RoboDK station: MESA_EJEMPLO.rdk

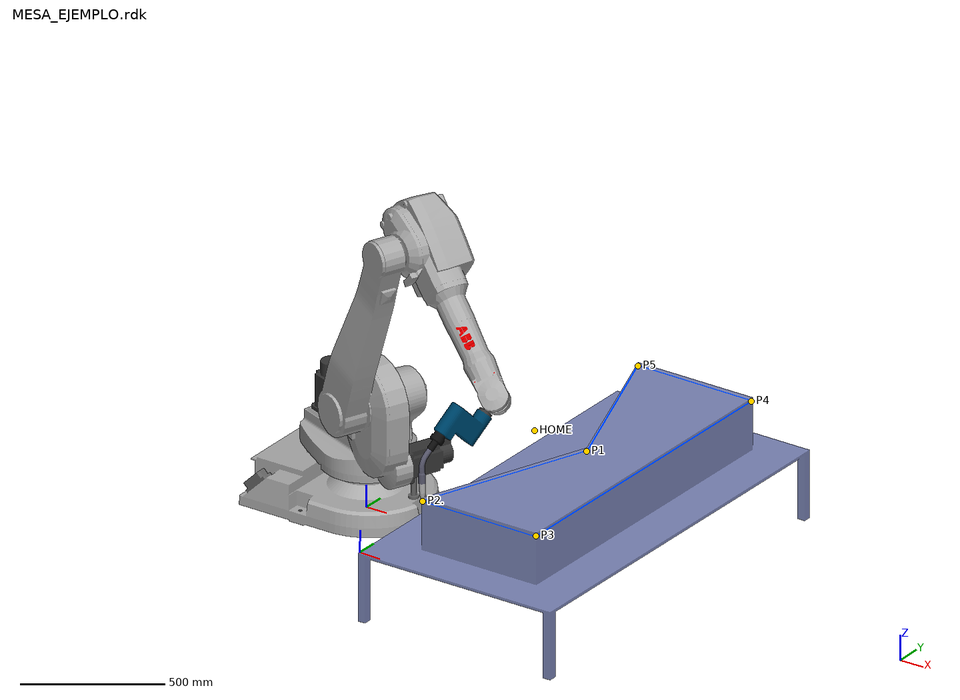
[picture v0: the station drawn from its stored meshes, robots at their saved joint values, targets as dots, program paths as lines]
Station MESA_EJEMPLO (saved by RoboDK 5.9.0). Poses are relative to the parent item; angles as X-Y-Z fixed-axis rotations.
  - frame ABB IRB 1600-6/1.45 Base at (0, 0, 0) mm
    - robot ABB IRB 1600-6/1.45: 6 axes, payload 6 kg, reach 1450 mm, repeatability 0.05 mm, weight 250 kg
        modified DH rows (alpha deg, a mm, theta deg, d mm): 0, 0, 0, 486.5; -90, 150, -90, 0; 0, 700, 0, 0; -90, 0, 0, 600; 90, 0, 0, 0; -90, 0, 180, 65
        joint limits [-180, -90, -245, -200, -115, -400] to [180, 120, 65, 200, 115, 400]; home [0, 0, 0, 0, 0, 0]; saved at [-21.7, 18.023, 24.268, -55.937, 59.398, 126.175]
      - tool Weld gun, TCP at (-4, 0, 371.3) mm, rotated rx 0 ry 45 rz 0 deg, size 299.9 x 60 x 318.3 mm
  - object mesa_ejemplo at (1300, -750, 0) mm, rotated rx 90 ry 0 rz 90 deg, size 1560 x 460 x 810 mm, geometry from mesa_ejemplo.IGS
  - frame Frame 2 at (500.14, -751.72, 267.07) mm, rotated rx -0.99 ry 1.63 rz 0.01 deg
    - target HOME (Cartesian target) at (159.13, 815.13, 203.86) mm, rotated rx 179.01 ry -0.28 rz 179.99 deg; joints [10.42, -21.045, 59.328, -38.186, 11.528, 45.27] of ABB IRB 1600-6/1.45
    - target P1 (Cartesian target) at (390.95, 796.79, 204.49) mm, rotated rx 179.01 ry -0.28 rz 179.99 deg; joints [4.664, 1.836, 43.09, -56.828, 3.804, 60.18] of ABB IRB 1600-6/1.45
    - target P2. (Cartesian target) at (152.66, 148.82, 186.18) mm, rotated rx 175.14 ry -1 rz 68.81 deg; joints [-21.7, 18.023, 24.268, -55.937, 59.398, 126.175] of ABB IRB 1600-6/1.45
    - target P3 (Cartesian target) at (630.12, 146.86, 199.37) mm, rotated rx 179.01 ry -0.28 rz 179.99 deg; joints [-35.771, 31.944, 0.147, 50.916, 30.958, -74.307] of ABB IRB 1600-6/1.45
    - target P4 (Cartesian target) at (630.36, 1444.09, 221.87) mm, rotated rx 179.01 ry -0.28 rz 179.99 deg; joints [39.829, 36.05, -7.07, -48.672, 35.634, 74.092] of ABB IRB 1600-6/1.45
    - target P5 (Cartesian target) at (150.28, 1447.38, 208.45) mm, rotated rx 179.01 ry -0.28 rz 179.99 deg; joints [63.12, 15.408, 26.322, -60.874, 44.224, 107.372] of ABB IRB 1600-6/1.45
    - target P1 (Cartesian target) at (390.95, 796.79, 204.49) mm, rotated rx 179.01 ry -0.28 rz 179.99 deg; joints [4.664, 1.836, 43.09, -56.828, 3.804, 60.18] of ABB IRB 1600-6/1.45
  - program Prog1 (8 instructions, listed below)
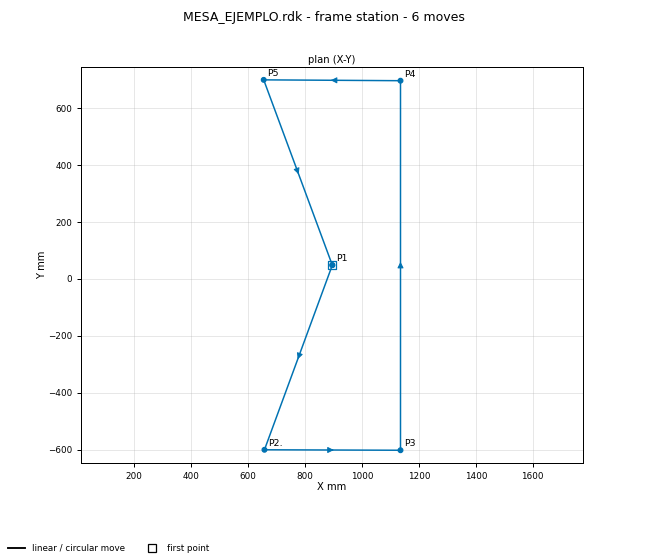
[picture p0: tool path of MESA_EJEMPLO.rdk in frame station, 6 of 6 moves have a stored position in this frame; points joined in program order, loops and branches not executed]

--- program Prog1 (robot ABB IRB 1600-6/1.45) ---
  Est. Ref.: Frame 2
  Est. herr: Weld gun
  MoveJ (P1)
  MoveL (P2.)
  MoveL (P3)
  MoveL (P4)
  MoveL (P5)
  MoveL (P1)
